{attribute addProperty BoxType "EL2502-0010-0020"}
{attribute addProperty Id "OvertemperatureBIT10.1251Short_Circuit_to_24_VBIT10.1254Feedback_PWMBIT10.1255Err_Start_TimeBIT10.1256"}
{attribute addProperty CRC "1505062968"}
{attribute addProperty SizeInBites "16"}
{attribute addProperty SizeInBytes "2"}
TYPE Status_59B57038 :
STRUCT
	{attribute addProperty Name "Overtemperature"}
	Overtemperature : BIT;
	{attribute 'hide'}
	reserve_1_BIT_0 : BIT;
	{attribute 'hide'}
	reserve_1_BIT_1 : BIT;
	{attribute addProperty Name "Short_Circuit_to_24_V"}
	Short_Circuit_to_24_V : BIT;
	{attribute addProperty Name "Feedback_PWM"}
	Feedback_PWM : BIT;
	{attribute addProperty Name "Err_Start_Time"}
	Err_Start_Time : BIT;
	{attribute 'hide'}
	reserve_2_BIT_0 : BIT;
	{attribute 'hide'}
	reserve_2_BIT_1 : BIT;
	{attribute 'hide'}
	reserve_3 : BYTE;
END_STRUCT
END_TYPE

(* stored: Version 1.2.0.0, ProductVersion 3.1.4024.9
   DUT Status_59B57038: Id {8f637300-03cd-4011-8c21-d0b9cc8684c2} *)
